FUNCTION_BLOCK DataPanel_MI_IXA (* Composite FB for boolean input data *)
  (* Standard: 61499-2; Description: Copyright (c) 2024 HR Agrartechnik GmbH This program and the accompanying materials are made available under the terms of the Eclipse Public License 2.0 which is available at https://www.eclipse.org/legal/epl-2.0/ SPDX-License-Identifier: EPL-2.0 *)
  (* Version 1.0, 2024-04-24, Franz Höpfinger, HR Agrartechnik GmbH *)
  PACKAGE DataPanel::io::MI::DI;
  IMPORT DataPanel::io::MI::const::MI;
  IMPORT eclipse4diac::core::TypeHash;
  IMPORT DataPanel::io::MI::DI::DataPanel_MI_DI::Invalid;
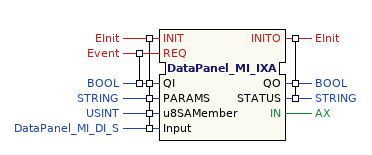
  EVENT_INPUT
    INIT : EInit WITH QI, PARAMS, u8SAMember, Input; (* Service Initialization *)
    REQ WITH QI; (* Service Request *)
  END_EVENT
  EVENT_OUTPUT
    INITO : EInit WITH QO, STATUS; (* Initialization Confirm *)
  END_EVENT
  VAR_INPUT
    QI : BOOL; (* Event Input Qualifier *)
    PARAMS : STRING; (* Service Parameters *)
    u8SAMember : USINT := MI::MI_00; (* Node SA 224..239 *)
    Input : DataPanel::io::MI::DI::DataPanel_MI_DI_S := Invalid; (* Identify the Input DigitalInput_5A..8B *)
  END_VAR
  VAR_OUTPUT
    QO : BOOL; (* Event Output Qualifier *)
    STATUS : STRING; (* Service Status *)
  END_VAR
  PLUGS
    IN : adapter::types::unidirectional::AX;
  END_PLUGS
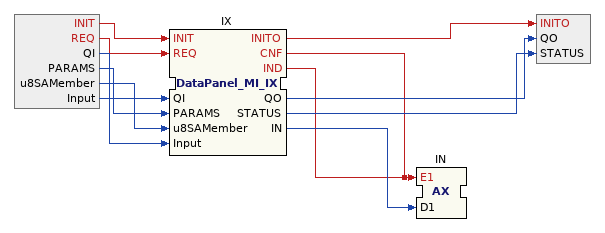
  FBS
    IX : DataPanel::io::MI::DI::DataPanel_MI_IX;
  END_FBS
  EVENT_CONNECTIONS
    INIT TO IX.INIT;
    IX.INITO TO INITO;
    IX.IND TO IN.E1;
    REQ TO IX.REQ;
    IX.CNF TO IN.E1;
  END_CONNECTIONS
  DATA_CONNECTIONS
    IX.IN TO IN.D1;
    QI TO IX.QI;
    PARAMS TO IX.PARAMS;
    IX.QO TO QO;
    IX.STATUS TO STATUS;
    u8SAMember TO IX.u8SAMember;
    Input TO IX.Input;
  END_CONNECTIONS
END_FUNCTION_BLOCK
